TYPE DUT_stBatchList :
STRUCT
	return_			: DINT;
	InputJson	: STRING(DB.MAX_STRING_SIZE);
	OutputJson	: STRING(DB.MAX_STRING_SIZE);
END_STRUCT
END_TYPE

(* stored: Version 1.1.0.1, ProductVersion 3.1.4024.15
   DUT DUT_stBatchList: Id {789d1f11-99f3-460e-a150-94a4371899bf} *)
